{attribute addProperty BoxType "EK1122-0000-0018"}
{attribute addProperty Id "Beckhoff_EJ1xxxsub_EK1100EK1100_179A0949162A_0001_EJ1100_0000_0018EJ1100_179A0949162A_0002_EJ1101_0022_0016EJ1101_6969C2248110.125"}
{attribute addProperty CRC "1564542346"}
{attribute addProperty SizeInBites "113"}
{attribute addProperty SizeInBytes "14.125"}
TYPE Beckhoff_EJ1xxxEK1122_5D41058A EXTENDS EK1122_179A0949 :
STRUCT
	{attribute addProperty Name "Beckhoff_EJ1xxxsub_EK1100"}
	Beckhoff_EJ1xxxsub_EK1100 : EK1100_179A0949;
	{attribute addProperty Name "A_0001_EJ1100_0000_0018"}
	A_0001_EJ1100_0000_0018 : EJ1100_179A0949;
	{attribute addProperty Name "A_0002_EJ1101_0022_0016"}
	A_0002_EJ1101_0022_0016 : EJ1101_6969C224;
END_STRUCT
END_TYPE

(* stored: Version 1.2.0.0, ProductVersion 3.1.4024.9
   DUT Beckhoff_EJ1xxxEK1122_5D41058A: Id {a1579d9a-660b-478e-8a95-8d7acc4b3692} *)
